TYPE ST_RejectReason_PK1_OUT2 :
STRUCT
	Reason	:STRING;
END_STRUCT
END_TYPE

(* stored: Version 1.1.0.1, ProductVersion 3.1.4024.13
   DUT ST_RejectReason_PK1_OUT2: Id {29211706-78b8-4859-8e8d-13131d164da0} *)
